{attribute 'GeneratedUsingTerminal: EL3751-0000-0020'}
{attribute addProperty BoxType "EL3751-0000-0020"}
{attribute addProperty Id "StatusAT %I*Status_543010BE7"}
{attribute addProperty CRC "2924134660"}
{attribute addProperty Size "7"}
TYPE PAI_Status_AE4AC104 :
STRUCT
	{attribute addProperty Name "Status"}
	Status AT %I* : Status_543010BE;
END_STRUCT
END_TYPE

(* stored: Version 1.2.0.0, ProductVersion 3.1.4024.9
   DUT PAI_Status_AE4AC104: Id {1ff164b6-f6d5-456c-be99-c5d04f09ada1} *)
